# B&R Automation Studio project TD52 (part 13)

### fintrf.h
```c
#if defined(WITH_COMMENTS)
/*
 * fintrf.h	- MATLAB/FORTRAN interface header file. This file
 *		  contains the declaration of the pointer type needed
 *		  by the MATLAB/FORTRAN interface.
 *
 * Copyright 1984-2008 The MathWorks, Inc.
 * All Rights Reserved.
 */
#endif
#if defined(__x86_64__) || defined(_M_AMD64) || defined(__amd64) || \
    defined(__sparcv9)  || defined(__ppc64__)
# define mwpointer integer*8
# define mwPointer integer*8
# define MWPOINTER INTEGER*8
#else
# define mwpointer integer*4
# define mwPointer integer*4
# define MWPOINTER INTEGER*4
#endif

#if defined(MX_COMPAT_32)
# define mwsize  integer*4
# define mwSize  integer*4
# define MWSIZE  INTEGER*4
# define mwindex integer*4
# define mwIndex integer*4
# define MWINDEX INTEGER*4
# define mwsignedindex integer*4
# define mwSignedIndex integer*4
# define MWSIGNEDINDEX INTEGER*4
#else
# define mwsize  mwpointer
# define mwSize  mwpointer
# define MWSIZE  MWPOINTER
# define mwindex mwpointer
# define mwIndex mwpointer
# define MWINDEX MWPOINTER
# define mwsignedindex mwpointer
# define mwSignedIndex mwpointer
# define MWSIGNEDINDEX MWPOINTER
#endif

#if defined(WITH_COMMENTS)
/*
 * Compatibility layer for MEX files using the 32-bit mxArray APIs
 */
#endif

#if defined(MX_COMPAT_32)

#define mxCalcSingleSubscript mxCalcSingleSubscript700
#define mxCreateCellArray mxCreateCellArray700
#define mxCreateCellMatrix mxCreateCellMatrix700
#define mxCreateCharArray mxCreateCharArray700
#define mxCreateCharMatrixFromStrings mxCreateCharMatrixFromStrs700
#define mxCreateDoubleMatrix mxCreateDoubleMatrix700
#define mxCreateNumericArray mxCreateNumericArray700
#define mxCreateNumericMatrix mxCreateNumericMatrix700
#define mxCreateSparse mxCreateSparse700
#define mxCreateStructArray mxCreateStructArray700
#define mxCreateStructMatrix mxCreateStructMatrix700
#define mxGetCell mxGetCell700
#define mxGetDimensions mxGetDimensions700
#define mxGetField mxGetField700
#define mxGetFieldByNumber mxGetFieldByNumber700
#define mxGetProperty mxGetProperty700
#define mxGetIr mxGetIr700
#define mxGetJc mxGetJc700
#define mxGetNumberOfDimensions mxGetNumberOfDimensions700
#define mxGetNzmax mxGetNzmax700
#define mxGetString mxGetString700
#define mxSetCell mxSetCell700
#define mxSetDimensions mxSetDimensions700
#define mxSetField mxSetField700
#define mxSetFieldByNumber mxSetFieldByNumber700
#define mxSetProperty mxSetProperty700
#define mxSetIr mxSetIr700
#define mxSetJc mxSetJc700
#define mxSetM mxSetM700
#define mxSetN mxSetN700
#define mxSetNzmax mxSetNzmax700
#define mxGetM mxGetM700
#define mxGetN mxGetN700
#define mxGetNumberOfElements mxGetNumberOfElements700
#define mxGetElementSize mxGetElementSize700
#define mxMalloc mxMalloc700
#define mxCalloc mxCalloc700
#define mxRealloc mxRealloc700
#define mxCopyReal4ToPtr mxCopyReal4ToPtr700
#define mxCopyPtrToReal4 mxCopyPtrToReal4700
#define mxCopyReal8ToPtr mxCopyReal8ToPtr700
#define mxCopyPtrToReal8 mxCopyPtrToReal8700
#define mxCopyCharacterToPtr mxCopyCharacterToPtr700
#define mxCopyPtrToCharacter mxCopyPtrToCharacter700
#define mxCopyInteger1ToPtr mxCopyInteger1ToPtr700
#define mxCopyPtrToInteger1 mxCopyPtrToInteger1700
#define mxCopyInteger2ToPtr mxCopyInteger2ToPtr700
#define mxCopyPtrToInteger2 mxCopyPtrToInteger2700
#define mxCopyInteger4ToPtr mxCopyInteger4ToPtr700
#define mxCopyPtrToInteger4 mxCopyPtrToInteger4700
#define mxCopyInteger8ToPtr mxCopyInteger8ToPtr700
#define mxCopyPtrToInteger8 mxCopyPtrToInteger8700
#define mxCopyPtrToPtrArray mxCopyPtrToPtrArray700
#define mxCopyComplex16ToPtr mxCopyComplex16ToPtr700
#define mxCopyPtrToComplex16 mxCopyPtrToComplex16700
#define mxCopyComplex8ToPtr mxCopyComplex8ToPtr700
#define mxCopyPtrToComplex8 mxCopyPtrToComplex8700
#define mxCopyMWIndexToPtr mxCopyMWIndexToPtr700
#define mxCopyPtrToMWIndex mxCopyPtrToMWIndex700
#define mxCreateCharMatrixFromStrs mxCreateCharMatrixFromStrs700
#define MXCALCSINGLESUBSCRIPT MXCALCSINGLESUBSCRIPT700
#define MXCREATECELLARRAY MXCREATECELLARRAY700
#define MXCREATECELLMATRIX MXCREATECELLMATRIX700
#define MXCREATECHARARRAY MXCREATECHARARRAY700
#define MXCREATECHARMATRIXFROMSTRINGS MXCREATECHARMATRIXFROMSTRS700
#define MXCREATEDOUBLEMATRIX MXCREATEDOUBLEMATRIX700
#define MXCREATENUMERICARRAY MXCREATENUMERICARRAY700
#define MXCREATENUMERICMATRIX MXCREATENUMERICMATRIX700
#define MXCREATESPARSE MXCREATESPARSE700
#define MXCREATESTRUCTARRAY MXCREATESTRUCTARRAY700
#define MXCREATESTRUCTMATRIX MXCREATESTRUCTMATRIX700
#define MXGETCELL MXGETCELL700
#define MXGETDIMENSIONS MXGETDIMENSIONS700
#define MXGETFIELD MXGETFIELD700
#define MXGETFIELDBYNUMBER MXGETFIELDBYNUMBER700
#define MXGETPROPERTY MXGETPROPERTY700
#define MXGETIR MXGETIR700
#define MXGETJC MXGETJC700
#define MXGETNUMBEROFDIMENSIONS MXGETNUMBEROFDIMENSIONS700
#define MXGETNZMAX MXGETNZMAX700
#define MXGETSTRING MXGETSTRING700
#define MXSETCELL MXSETCELL700
#define MXSETDIMENSIONS MXSETDIMENSIONS700
#define MXSETFIELD MXSETFIELD700
#define MXSETFIELDBYNUMBER MXSETFIELDBYNUMBER700
#define MXSETPROPERTY MXSETPROPERTY700
#define MXSETIR MXSETIR700
#define MXSETJC MXSETJC700
#define MXSETM MXSETM700
#define MXSETN MXSETN700
#define MXSETNZMAX MXSETNZMAX700
#define MXGETM MXGETM700
#define MXGETN MXGETN700
#define MXGETNUMBEROFELEMENTS MXGETNUMBEROFELEMENTS700
#define MXGETELEMENTSIZE MXGETELEMENTSIZE700
#define MXMALLOC MXMALLOC700
#define MXCALLOC MXCALLOC700
#define MXREALLOC MXREALLOC700
#define MXCOPYREAL4TOPTR MXCOPYREAL4TOPTR700
#define MXCOPYPTRTOREAL4 MXCOPYPTRTOREAL4700
#define MXCOPYREAL8TOPTR MXCOPYREAL8TOPTR700
#define MXCOPYPTRTOREAL8 MXCOPYPTRTOREAL8700
#define MXCOPYCHARACTERTOPTR MXCOPYCHARACTERTOPTR700
#define MXCOPYPTRTOCHARACTER MXCOPYPTRTOCHARACTER700
#define MXCOPYINTEGER1TOPTR MXCOPYINTEGER1TOPTR700
#define MXCOPYPTRTOINTEGER1 MXCOPYPTRTOINTEGER1700
#define MXCOPYINTEGER2TOPTR MXCOPYINTEGER2TOPTR700
#define MXCOPYPTRTOINTEGER2 MXCOPYPTRTOINTEGER2700
#define MXCOPYINTEGER4TOPTR MXCOPYINTEGER4TOPTR700
#define MXCOPYPTRTOINTEGER4 MXCOPYPTRTOINTEGER4700
#define MXCOPYINTEGER8TOPTR MXCOPYINTEGER8TOPTR700
#define MXCOPYPTRTOINTEGER8 MXCOPYPTRTOINTEGER8700
#define MXCOPYPTRTOPTRARRAY MXCOPYPTRTOPTRARRAY700
#define MXCOPYCOMPLEX16TOPTR MXCOPYCOMPLEX16TOPTR700
#define MXCOPYPTRTOCOMPLEX16 MXCOPYPTRTOCOMPLEX16700
#define MXCOPYCOMPLEX8TOPTR MXCOPYCOMPLEX8TOPTR700
#define MXCOPYPTRTOCOMPLEX8 MXCOPYPTRTOCOMPLEX8700
#define MXCOPYMWINDEXTOPTR MXCOPYMWINDEXTOPTR700
#define MXCOPYPTRTOMWINDEX MXCOPYPTRTOMWINDEX700
#define MXCREATECHARMATRIXFROMSTRS MXCREATECHARMATRIXFROMSTRS700
#define mxcalcsinglesubscript mxcalcsinglesubscript700
#define mxcreatecellarray mxcreatecellarray700
#define mxcreatecellmatrix mxcreatecellmatrix700
#define mxcreatechararray mxcreatechararray700
#define mxcreatecharmatrixfromstrings mxcreatecharmatrixfromstrs700
#define mxcreatedoublematrix mxcreatedoublematrix700
#define mxcreatenumericarray mxcreatenumericarray700
#define mxcreatenumericmatrix mxcreatenumericmatrix700
#define mxcreatesparse mxcreatesparse700
#define mxcreatestructarray mxcreatestructarray700
#define mxcreatestructmatrix mxcreatestructmatrix700
#define mxgetcell mxgetcell700
#define mxgetdimensions mxgetdimensions700
#define mxgetfield mxgetfield700
#define mxgetfieldbynumber mxgetfieldbynumber700
#define mxgetproperty mxgetproperty700
#define mxgetir mxgetir700
#define mxgetjc mxgetjc700
#define mxgetnumberofdimensions mxgetnumberofdimensions700
#define mxgetnzmax mxgetnzmax700
#define mxgetstring mxgetstring700
#define mxsetcell mxsetcell700
#define mxsetdimensions mxsetdimensions700
#define mxsetfield mxsetfield700
#define mxsetfieldbynumber mxsetfieldbynumber700
#define mxsetproperty mxsetproperty700
#define mxsetir mxsetir700
#define mxsetjc mxsetjc700
#define mxsetm mxsetm700
#define mxsetn mxsetn700
#define mxsetnzmax mxsetnzmax700
#define mxgetm mxgetm700
#define mxgetn mxgetn700
#define mxgetnumberofelements mxgetnumberofelements700
#define mxgetelementsize mxgetelementsize700
#define mxmalloc mxmalloc700
#define mxcalloc mxcalloc700
#define mxrealloc mxrealloc700
#define mxcopyreal4toptr mxcopyreal4toptr700
#define mxcopyptrtoreal4 mxcopyptrtoreal4700
#define mxcopyreal8toptr mxcopyreal8toptr700
#define mxcopyptrtoreal8 mxcopyptrtoreal8700
#define mxcopycharactertoptr mxcopycharactertoptr700
#define mxcopyptrtocharacter mxcopyptrtocharacter700
#define mxcopyinteger1toptr mxcopyinteger1toptr700
#define mxcopyptrtointeger1 mxcopyptrtointeger1700
#define mxcopyinteger2toptr mxcopyinteger2toptr700
#define mxcopyptrtointeger2 mxcopyptrtointeger2700
#define mxcopyinteger4toptr mxcopyinteger4toptr700
#define mxcopyptrtointeger4 mxcopyptrtointeger4700
#define mxcopyinteger8toptr mxcopyinteger8toptr700
#define mxcopyptrtointeger8 mxcopyptrtointeger8700
#define mxcopyptrtoptrarray mxcopyptrtoptrarray700
#define mxcopycomplex16toptr mxcopycomplex16toptr700
#define mxcopyptrtocomplex16 mxcopyptrtocomplex16700
#define mxcopycomplex8toptr mxcopycomplex8toptr700
#define mxcopyptrtocomplex8 mxcopyptrtocomplex8700
#define mxcopymwindextoptr mxcopymwindextoptr700
#define mxcopyptrtomwindex mxcopyptrtomwindex700
#define mxcreatecharmatrixfromstrs mxcreatecharmatrixfromstrs700

#else

#ifndef __linux
#define mxCalcSingleSubscript mxCalcSingleSubscript730
#define mxCreateCellArray mxCreateCellArray730
#define mxCreateCellMatrix mxCreateCellMatrix730
#define mxCreateCharArray mxCreateCharArray730
#define mxCreateCharMatrixFromStrings mxCreateCharMatrixFromStrs730
#define mxCreateDoubleMatrix mxCreateDoubleMatrix730
#define mxCreateNumericArray mxCreateNumericArray730
#define mxCreateNumericMatrix mxCreateNumericMatrix730
#define mxCreateSparse mxCreateSparse730
#define mxCreateStructArray mxCreateStructArray730
#define mxCreateStructMatrix mxCreateStructMatrix730
#define mxGetCell mxGetCell730
#define mxGetDimensions mxGetDimensions730
#define mxGetField mxGetField730
#define mxGetFieldByNumber mxGetFieldByNumber730
#define mxGetProperty mxGetProperty730
#define mxGetIr mxGetIr730
#define mxGetJc mxGetJc730
#define mxGetNumberOfDimensions mxGetNumberOfDimensions730
#define mxGetNzmax mxGetNzmax730
#define mxGetString mxGetString730
#define mxSetCell mxSetCell730
#define mxSetDimensions mxSetDimensions730
#define mxSetField mxSetField730
#define mxSetFieldByNumber mxSetFieldByNumber730
#define mxSetProperty mxSetProperty730
#define mxSetIr mxSetIr730
#define mxSetJc mxSetJc730
#define mxSetM mxSetM730
#define mxSetN mxSetN730
#define mxSetNzmax mxSetNzmax730
#define mxGetM mxGetM730
#define mxGetN mxGetN730
#define mxGetNumberOfElements mxGetNumberOfElements730
#define mxGetElementSize mxGetElementSize730
#define mxMalloc mxMalloc730
#define mxCalloc mxCalloc730
#define mxRealloc mxRealloc730
#define mxCopyReal4ToPtr mxCopyReal4ToPtr730
#define mxCopyPtrToReal4 mxCopyPtrToReal4730
#define mxCopyReal8ToPtr mxCopyReal8ToPtr730
#define mxCopyPtrToReal8 mxCopyPtrToReal8730
#define mxCopyCharacterToPtr mxCopyCharacterToPtr730
#define mxCopyPtrToCharacter mxCopyPtrToCharacter730
#define mxCopyInteger1ToPtr mxCopyInteger1ToPtr730
#define mxCopyPtrToInteger1 mxCopyPtrToInteger1730
#define mxCopyInteger2ToPtr mxCopyInteger2ToPtr730
#define mxCopyPtrToInteger2 mxCopyPtrToInteger2730
#define mxCopyInteger4ToPtr mxCopyInteger4ToPtr730
#define mxCopyPtrToInteger4 mxCopyPtrToInteger4730
#define mxCopyInteger8ToPtr mxCopyInteger8ToPtr730
#define mxCopyPtrToInteger8 mxCopyPtrToInteger8730
#define mxCopyPtrToPtrArray mxCopyPtrToPtrArray730
#define mxCopyComplex16ToPtr mxCopyComplex16ToPtr730
#define mxCopyPtrToComplex16 mxCopyPtrToComplex16730
#define mxCopyComplex8ToPtr mxCopyComplex8ToPtr730
#define mxCopyPtrToComplex8 mxCopyPtrToComplex8730
#define mxCopyMWIndexToPtr mxCopyMWIndexToPtr730
#define mxCopyPtrToMWIndex mxCopyPtrToMWIndex730
#define mxCreateCharMatrixFromStrs mxCreateCharMatrixFromStrs730
#define MXCALCSINGLESUBSCRIPT MXCALCSINGLESUBSCRIPT730
#define MXCREATECELLARRAY MXCREATECELLARRAY730
#define MXCREATECELLMATRIX MXCREATECELLMATRIX730
#define MXCREATECHARARRAY MXCREATECHARARRAY730
#define MXCREATECHARMATRIXFROMSTRINGS MXCREATECHARMATRIXFROMSTRS730
#define MXCREATEDOUBLEMATRIX MXCREATEDOUBLEMATRIX730
#define MXCREATENUMERICARRAY MXCREATENUMERICARRAY730
#define MXCREATENUMERICMATRIX MXCREATENUMERICMATRIX730
#define MXCREATESPARSE MXCREATESPARSE730
#define MXCREATESTRUCTARRAY MXCREATESTRUCTARRAY730
#define MXCREATESTRUCTMATRIX MXCREATESTRUCTMATRIX730
#define MXGETCELL MXGETCELL730
#define MXGETDIMENSIONS MXGETDIMENSIONS730
#define MXGETFIELD MXGETFIELD730
#define MXGETFIELDBYNUMBER MXGETFIELDBYNUMBER730
#define MXGETPROPERTY MXGETPROPERTY730
#define MXGETIR MXGETIR730
#define MXGETJC MXGETJC730
#define MXGETNUMBEROFDIMENSIONS MXGETNUMBEROFDIMENSIONS730
#define MXGETNZMAX MXGETNZMAX730
#define MXGETSTRING MXGETSTRING730
#define MXSETCELL MXSETCELL730
#define MXSETDIMENSIONS MXSETDIMENSIONS730
#define MXSETFIELD MXSETFIELD730
#define MXSETFIELDBYNUMBER MXSETFIELDBYNUMBER730
#define MXSETPROPERTY MXSETPROPERTY730
#define MXSETIR MXSETIR730
#define MXSETJC MXSETJC730
#define MXSETM MXSETM730
#define MXSETN MXSETN730
#define MXSETNZMAX MXSETNZMAX730
#define MXGETM MXGETM730
#define MXGETN MXGETN730
#define MXGETNUMBEROFELEMENTS MXGETNUMBEROFELEMENTS730
#define MXGETELEMENTSIZE MXGETELEMENTSIZE730
#define MXMALLOC MXMALLOC730
#define MXCALLOC MXCALLOC730
#define MXREALLOC MXREALLOC730
#define MXCOPYREAL4TOPTR MXCOPYREAL4TOPTR730
#define MXCOPYPTRTOREAL4 MXCOPYPTRTOREAL4730
#define MXCOPYREAL8TOPTR MXCOPYREAL8TOPTR730
#define MXCOPYPTRTOREAL8 MXCOPYPTRTOREAL8730
#define MXCOPYCHARACTERTOPTR MXCOPYCHARACTERTOPTR730
#define MXCOPYPTRTOCHARACTER MXCOPYPTRTOCHARACTER730
#define MXCOPYINTEGER1TOPTR MXCOPYINTEGER1TOPTR730
#define MXCOPYPTRTOINTEGER1 MXCOPYPTRTOINTEGER1730
#define MXCOPYINTEGER2TOPTR MXCOPYINTEGER2TOPTR730
#define MXCOPYPTRTOINTEGER2 MXCOPYPTRTOINTEGER2730
#define MXCOPYINTEGER4TOPTR MXCOPYINTEGER4TOPTR730
#define MXCOPYPTRTOINTEGER4 MXCOPYPTRTOINTEGER4730
#define MXCOPYINTEGER8TOPTR MXCOPYINTEGER8TOPTR730
#define MXCOPYPTRTOINTEGER8 MXCOPYPTRTOINTEGER8730
#define MXCOPYPTRTOPTRARRAY MXCOPYPTRTOPTRARRAY730
#define MXCOPYCOMPLEX16TOPTR MXCOPYCOMPLEX16TOPTR730
#define MXCOPYPTRTOCOMPLEX16 MXCOPYPTRTOCOMPLEX16730
#define MXCOPYCOMPLEX8TOPTR MXCOPYCOMPLEX8TOPTR730
#define MXCOPYPTRTOCOMPLEX8 MXCOPYPTRTOCOMPLEX8730
#define MXCOPYMWINDEXTOPTR MXCOPYMWINDEXTOPTR730
#define MXCOPYPTRTOMWINDEX MXCOPYPTRTOMWINDEX730
#define MXCREATECHARMATRIXFROMSTRS MXCREATECHARMATRIXFROMSTRS730
#define mxcalcsinglesubscript mxcalcsinglesubscript730
#define mxcreatecellarray mxcreatecellarray730
#define mxcreatecellmatrix mxcreatecellmatrix730
#define mxcreatechararray mxcreatechararray730
#define mxcreatecharmatrixfromstrings mxcreatecharmatrixfromstrs730
#define mxcreatedoublematrix mxcreatedoublematrix730
#define mxcreatenumericarray mxcreatenumericarray730
#define mxcreatenumericmatrix mxcreatenumericmatrix730
#define mxcreatesparse mxcreatesparse730
#define mxcreatestructarray mxcreatestructarray730
#define mxcreatestructmatrix mxcreatestructmatrix730
#define mxgetcell mxgetcell730
#define mxgetdimensions mxgetdimensions730
#define mxgetfield mxgetfield730
#define mxgetfieldbynumber mxgetfieldbynumber730
#define mxgetproperty mxgetproperty730
#define mxgetir mxgetir730
#define mxgetjc mxgetjc730
#define mxgetnumberofdimensions mxgetnumberofdimensions730
#define mxgetnzmax mxgetnzmax730
#define mxgetstring mxgetstring730
#define mxsetcell mxsetcell730
#define mxsetdimensions mxsetdimensions730
#define mxsetfield mxsetfield730
#define mxsetfieldbynumber mxsetfieldbynumber730
#define mxsetproperty mxsetproperty730
#define mxsetir mxsetir730
#define mxsetjc mxsetjc730
#define mxsetm mxsetm730
#define mxsetn mxsetn730
#define mxsetnzmax mxsetnzmax730
#define mxgetm mxgetm730
#define mxgetn mxgetn730
#define mxgetnumberofelements mxgetnumberofelements730
#define mxgetelementsize mxgetelementsize730
#define mxmalloc mxmalloc730
#define mxcalloc mxcalloc730
#define mxrealloc mxrealloc730
#define mxcopyreal4toptr mxcopyreal4toptr730
#define mxcopyptrtoreal4 mxcopyptrtoreal4730
#define mxcopyreal8toptr mxcopyreal8toptr730
#define mxcopyptrtoreal8 mxcopyptrtoreal8730
#define mxcopycharactertoptr mxcopycharactertoptr730
#define mxcopyptrtocharacter mxcopyptrtocharacter730
#define mxcopyinteger1toptr mxcopyinteger1toptr730
#define mxcopyptrtointeger1 mxcopyptrtointeger1730
#define mxcopyinteger2toptr mxcopyinteger2toptr730
#define mxcopyptrtointeger2 mxcopyptrtointeger2730
#define mxcopyinteger4toptr mxcopyinteger4toptr730
#define mxcopyptrtointeger4 mxcopyptrtointeger4730
#define mxcopyinteger8toptr mxcopyinteger8toptr730
#define mxcopyptrtointeger8 mxcopyptrtointeger8730
#define mxcopyptrtoptrarray mxcopyptrtoptrarray730
#define mxcopycomplex16toptr mxcopycomplex16toptr730
#define mxcopyptrtocomplex16 mxcopyptrtocomplex16730
#define mxcopycomplex8toptr mxcopycomplex8toptr730
#define mxcopyptrtocomplex8 mxcopyptrtocomplex8730
#define mxcopymwindextoptr mxcopymwindextoptr730
#define mxcopyptrtomwindex mxcopyptrtomwindex730
#define mxcreatecharmatrixfromstrs mxcreatecharmatrixfromstrs730
#endif

#endif
```

### fixedpoint.h
```c
#include "fixpoint_spec.hpp"
/* Copyright 1994-2010 The MathWorks, Inc.
 * $Revision: 1.1.8.1 $
 * $Date: 2010/12/15 17:39:58 $
 */

#ifdef SUPPORTS_PRAGMA_ONCE
#pragma once
#endif

#ifndef fix_published_intro_h
#define fix_published_intro_h

/* Abstract:
 *
 * The primary motivation of this header file is to allow customers to
 * write C language S-functions that support fixed-point data types.  However,
 * the API in this header extends beyond fixed-point and includes support for
 * standard floating point and integer data types.
 *
 * This header contains definitions and prototypes for use in creating
 * Simulink S-functions that can process a wide variety of data types.
 * These data types include the Simulink builtin data types,
 *     double        single
 *     uint8         int8
 *     uint16        int16
 *     uint32        int32
 * all the MathWorks defined fixed-point data types such as
 *     sfix16_En15
 *     ufix32_En16
 *     ufix128
 *     sfix37_S3_B5
 * and the versions of data types obtained when Data Type Override is set
 * to Scaled Doubles such as
 *     flts16
 *     flts16_En15
 *     fltu32_S3_B5
 *
 * This header file contains functions and definitions that allow S-functions
 * to determine which of these data types an input port or output port is
 * using.  The S-function can also specify which of these data types should
 * be used for an input, output, DWork state, or Runtime Parameter.  The
 * information required to properly read to and write from different variables
 * of each data type is given.
 */

/* Note on License Design:
 *
 * The following comments are simply an attempt to clarify the License Design
 * so that authors can write better S-functions.
 * As of
 *      Release 13
 *      Simulink 5.0
 *      Fixed-Point Blockset 4.0
 * all the blocks from Fixed-Point Blockset were merged into Simulink.  All
 * the blocks are installed even if a user does not have a Fixed-Point License.
 * Simulink customers can use all the blocks with any builtin data types that a
 * block supports.  If all the blocks in a model are only using builtin data
 * types and the Min-Max-Overflow Logging Mode is set to Force Off, then a
 * Fixed-Point License is NOT required.  If any block in a model is "actively"
 * using a non-builtin fixed-point data type or is actively logging Min-Max and/or
 * Overflow information, then a Fixed-Point License will be required for the
 * remainder of that Matlab session.
 *   Even if blocks in a model are configured to have fixed-point signals and/or
 * configured to log Min-Max-Overflow information, then simply loading, viewing,
 * editing, or saving a model should not trigger active use.  Actions such as
 * Update Diagram, Simulation, and Code Generation from such a model are active
 * use and would cause a Fixed-Point License to be checked out.
 *   S-functions written using the API in this header file should be able to
 * follow this license design.  For example, suppose an S-function is written
 * so that it can handle any builtin or fixed-point data type.  Suppose in a
 * particular model, this S-function is processing just builtin data types such
 * as double, single, uint8, or int32.  That use case would not trigger a
 * Fixed-Point License to be checked out.  Suppose in a different model,
 * the S-function was processing non-builtin fixed-point data types.  That use,
 * like any other use of fixed-point data types, would cause a Fixed-Point
 * License to be checked out.
 *   The key pitfall S-function authors must guard against is registering
 * a fixed-point data type when a model is simply being loaded or viewed.  In
 * Simulink jargon, loading or opening a model or sub-system is a
 * "Sizes Call Only."  The Simulink S-function API provides a way to detect a
 * "Sizes Call Only", so by careful programming, an S-function author can avoid
 * Fixed-Point License problems when a user is simply loading or viewing a model.
 */

/* Simulink supports fixed-point data types with any number of bits from
 *    1 to FXP_MAX_BITS for unsigned numbers and
 *    2 to FXP_MAX_BITS for signed numbers.
 * The API in this header file treats pure integers just like
 * any other fixed-point numbers.  Pure integers just happen
 * to have trivial scaling.  The 6 standard Simulink integer
 * types uint8, int8, uint16, int16, uint32, and int32 are not
 * exceptions.  They are treated like fixed-point numbers
 * that happened to have trivial scaling and happened to have
 * 8, 16, or 32 bits.  The same API applies.
 *   Simulink builtin integers are special only in that they do
 * not trigger the need for a Fixed-Point License.
 *
 * The number of bits used to represent a signal in simulation
 * may be more than the number specified.  In this case, the
 * signals will be emulated inside various sized containers
 * according to the following rules.  For 32 or fewer bits, the
 * rules are simple.  For 32 or fewer bits, the container is a
 * scalar integer type directly understood by the compiler.  The
 * case of using a scalar integer type is classified as single-word.
 * The three cases with 32 or fewer bits are shown by a table.
 *
 *   Specified Bits       Container Bits   Container typedef
 *    1 to  8              8               int8_T  or uint8_T
 *    9 to 16             16               int16_T or uint16_T
 *   17 to 32             32               int32_T or uint32_T
 *
 * For 33 or more bits, the rules are more complicated and can
 * depend on the model, the Matlab Host, the current target
 * for code generation, and the version of Simulink Fixed Point
 * being used.  Signals with 33 or more bits will either be stored
 * using a single-word
 * container with more than 32 bits or will be stored using a
 * multi-word representation.
 *
 * All multi-word representations will follow a general form.
 *
 * typedef struct {
 *     SOME_UNSIGNED_CHUNK_TYPE chunks[ NUM_CHUNKS_FOR_M_BITS ];
 * } (u)intM_T
 *
 * The chunk at index zero will hold the least significant bits, and
 * the highest index will hold the most significant bits.
 *
 * Whether single-word or multi-word is used can depend on
 * the model, the Matlab Host, the current
 * target for code generation, and the version of Simulink Fixed Point.
 * The specific type used for SOME_UNSIGNED_CHUNK_TYPE can also vary depending
 * on the model, the Matlab Host, the current target for code generation,
 * and the version of Simulink Fixed Point.
 *
 * To be portable, sfunctions that are intended to support fixed-point
 * signals with more than 32 bits must react to container variations
 * at runtime.  The most general way to do this is to use the interfaces
 * for getting and setting "bit-regions" provided by this header.
 * To support use of code optimized to a specific additional APIs
 * are provided that can query the current properties of a data type.
 * However, sfunction authors need to be aware the properties of a data
 * type can vary depending on
 * the model, the Matlab Host, the current
 * target for code generation, and the version of Simulink Fixed Point.
 * A robustly written sfunction will need to check the properties at runtime
 * at least once after update diagram has started.  The most portable sfunctions
 * will be written so that they can use an optimized case if possible or
 * switch to general bit-region case if necessary.  At the very least,
 * a robust sfunction will need to gracefully set an error if does not
 * have a case that supports the current memory layout.  Keep in mind that
 * supporting every specific case for the current release of Simulink Fixed Point
 * does not guarantee that every specific case in a future release will be
 * covered.  For this reason, it is best to have bit-region case or at
 * the very least gracefully error if needed.
 *
 * For signed numbers, the bit encoding format is always
 * two's complement.
 *
 * When the specified number of bits is less than the size of
 * the container, the desired bits are always stored in the
 * least significant part of the container.  Any "unused" bits
 * are in the most significant part of the container.
 *
 * For both single word case and multiword cases, any unused bits
 * must be set to a sign extension.  If the data type is
 * an unsigned number, then obviously, the number is always
 * nonnegative so the (implicit) sign bit is zero.  For unsigned
 * data types, all unused bits must always be cleared to zero.
 *    If the data type is a signed number, then the sign bit is
 * one for strictly negative numbers and zero otherwise.  If
 * the stored integer is negative, then all unused bits must be
 * set to one.  If the stored integer is positive, then all
 * unused bits must be cleared to zero.
 *
 * Simulink also supports two builtin floating point data types.
 * These are the standard floating point singles and doubles.
 *
 * Simulink also supports a data type category that is a hybrid
 * between floating-point and fixed-point.  This category is
 * called ScaledDouble.  ScaledDouble cases occur when
 * an individual block is configured to have a fixed-point
 * output, but the system it lives in has its Data Type Override
 * setting for a system is set to Scaled Doubles.  The
 * resulting data type has the scaling the fixed-point
 * specification, but stores its output using floating
 * point doubles.  Storing in a double means that overflow
 * and precision issues are almost always eliminated. Removing the
 * range and precision issues is very useful for benchmarking, testing,
 * and debugging.
 *   ScaledDouble data types contain information
 * signedness and number of bits of what their non-overrided data
 * types would have been.  This is useful for information for other
 * portions of the model that are not being debugged with Data Type
 * Override.
 */

#endif /* fix_published_intro_h */
/* Copyright 1994-2010 The MathWorks, Inc.
 * $Revision: 1.1.6.1 $
 * $Date: 2010/06/15 00:02:53 $
 */

#ifdef SUPPORTS_PRAGMA_ONCE
#pragma once
#endif

#ifndef fxplimits_h
#define fxplimits_h

#define FXP_MAX_BITS 128

#endif /* fxplimits_h */
/* Copyright 1994-2010 The MathWorks, Inc.
 * $Revision: 1.1.6.1 $
 * $Date: 2010/06/15 00:02:51 $
 */

#ifdef SUPPORTS_PRAGMA_ONCE
#pragma once
#endif

#ifndef fxpchunkarrary_h
#define fxpchunkarrary_h

typedef uint32_T FXP_CHUNK_T;

#define FXP_BITS_PER_CHUNK 32

#define FXP_NUM_CHUNKS ( FXP_MAX_BITS / FXP_BITS_PER_CHUNK )

#define FXP_INDEX_LEAST_SIGNIFICANT_CHUNK 0

#define FXP_INDEX_MOST_SIGNIFICANT_CHUNK  ( FXP_NUM_CHUNKS - 1 )

#define FXP_ALL_ONES_CHUNK 0xFFFFFFFFul

typedef struct fxpChunkArray_tag
{
    FXP_CHUNK_T chunk[ FXP_NUM_CHUNKS ];

} fxpChunkArray;

#endif /* fxpchunkarrary_h */
/* Copyright 1994-2010 The MathWorks, Inc.
 * $Revision: 1.1.8.1 $
 * $Date: 2010/12/15 17:40:00 $
 */

#ifdef SUPPORTS_PRAGMA_ONCE
#pragma once
#endif

#ifndef fxpsimulinkscalingintro_h
#define fxpsimulinkscalingintro_h

/* Simulink Scaling
 *
 * Simulink data types support scaling.  The Fixed-Point User's Guide
 * presents the following general formula.
 *
 *    V = S * Q + B
 *
 * where
 *
 *    V is the Real World Value in the engineering units of choice
 *    Q is the called the Stored Integer Value.  It is the raw value
 *      stored in the digital hardware.  Despite the name Q can use
 *      an integer or a floating point format.
 *    S is the Slope.  For clarity, this is also called the Total-Slope
 *    B is the Bias
 *
 * The Total-Slope is often decomposed into two parts.
 *
 *    S = F * 2^E
 *
 * where
 *
 *   1. <= F < 2.0
 *
 *    F is the Fractional Slope
 *    E is the Fixed Exponent, E is always an integer.
 *
 * If
 *    B == 0.0
 * and
 *    F == 1.0
 * then
 * there is a clean binary point interpretation.
 *
 *    Fraction Length = -1 * Fixed Exponent
 *
 * For example, if
 *    S == 0.125
 *    B == 0.0
 * then
 *    F == 1.0
 *    E == -3
 * so
 *    Fraction Length = 3
 * therefore, this data type has 3 bits to the right of the
 * binary point.
 *
 * The concept of scaling is most useful for fixed-point cases, but
 * it does generalize to all the scalar numeric data types.  For
 * floating point doubles and singles and for pure integers,
 * the scaling is trivial
 *    B == 0
 *    S == 1
 *    F == 1
 *    E == 0
 *    Fraction Length == 0
 * The access methods to get scaling information can be used
 * for all the data types, they just return trivial values
 * when the scaling is trivial.
 */

#endif /* fxpsimulinkscalingintro_h */
/* Copyright 1994-2010 The MathWorks, Inc.
 * $Revision: 1.1.6.1 $
 * $Date: 2010/06/15 00:02:55 $
 */

#ifdef SUPPORTS_PRAGMA_ONCE
#pragma once
#endif

#ifndef fxpmodeoverflow_h
#define fxpmodeoverflow_h

/* The enums specify the overflow handling modes supported by most fixed-point
 * math functions.
 */
typedef enum fxpModeOverflow_tag {
  FXP_OVERFLOW_WRAP = 0, /* must be zero */
  FXP_OVERFLOW_SATURATE

} fxpModeOverflow;

#endif /* fxpmodeoverflow_h */
/* Copyright 1994-2010 The MathWorks, Inc.
 * $Revision: 1.1.6.1 $
 * $Date: 2010/06/15 00:02:57 $
 */

#ifdef SUPPORTS_PRAGMA_ONCE
#pragma once
#endif

#ifndef fxpmoderounding_h
#define fxpmoderounding_h

/* The enums specify the rounding modes supported by most fixed-point
 * math functions.
 */
typedef enum fxpModeRounding_tag {
  FXP_ROUND_ZERO = 0, /* must be zero */
  FXP_ROUND_NEAR,
  FXP_ROUND_CEIL,
  FXP_ROUND_FLOOR,
  FXP_ROUND_SIMPLEST,
  FXP_ROUND_NEAR_ML, /* Round -x.5 to -(x+1) not -x so as to match MATLAB. */
  FXP_ROUND_CONVERGENT
} fxpModeRounding;

#define FXP_ROUND_METHOD_COUNT ((FXP_ROUND_CONVERGENT)+1)

#endif /* fxpmoderounding_h */
/* Copyright 1994-2010 The MathWorks, Inc.
 * $Revision: 1.1.6.1 $
 * $Date: 2010/06/15 00:02:59 $
 */

#ifdef SUPPORTS_PRAGMA_ONCE
#pragma once
#endif

#ifndef fix_published_fxpOverflowLogs_h
#define fix_published_fxpOverflowLogs_h

/* Overflow logging structure
 *
 * Some fixed-point math functions accept a pointer to this structure.
 * These functions will initialize each of the event counts to zero.  Then
 * the functions will carryout the requested math operations.  Each
 * time an event is detect during the math operation the appropriate
 * count will be incremented.  The increment operations makes sure
 * the count does not overflow to zero; it will saturate to the upper limit.
 *
 * For example, suppose a fixed-point conversion function is called. Suppose,
 * one overflow occurred during the conversion.  After the function return,
 * the memory pointed to be overflow logging structure pointer would indicate
 * one overflow, zero saturations, and zero divide-by-zeros.
 */
typedef struct fxpOverflowLogs_tag
{
      int OverflowOccurred;
      int SaturationOccurred;
      int DivisionByZeroOccurred;

} fxpOverflowLogs;

#endif /* fix_published_fxpOverflowLogs_h */
/* Copyright 1994-2011 The MathWorks, Inc.
 *
 *
 */

#ifdef SUPPORTS_PRAGMA_ONCE
#pragma once
#endif

#ifndef fix_published_sfun_api_h
#define fix_published_sfun_api_h

/* Function: ssRegisterDataTypeFxpBinaryPoint ===============================
 *
 * This function fully registers a fixed-point data type with Simulink and
 * returns a Data Type Id.  Unlike the standard Simulink function,
 * ssRegisterDataType, additional registration steps do not need to be taken
 * and should not be taken.  The returned Data Type Id can be used to specify
 * the data types of input ports, output ports, RunTimeParameters, and DWork
 * states.  The Data Type Id can also be used with all the standard
 * data type access methods in simstruc.h such as ssGetDataTypeSize.
 *
 * The input arguments are
 *    isSigned              TRUE if signed, FALSE if unsigned
 *    wordLength            total number of bits including any sign bit
 *    fractionLength        number of bit to right of binary point
 *    obeyDataTypeOverride  if FALSE ignore system's setting for Data Type Override
 *                          if TRUE obey Data Type Override setting, depending
 *                          on Data Type Override, resulting data type could be
 *                          True Double, True Single, Scaled Double, or the
 *                          requested fixed point type.
 *
 * Cautions:
 *
 * 1) If the registered data type is not one of the builtin data types, then
 * a Fixed-Point License will be checked out.  To prevent, a Fixed-Point
 * License from being checked out when a user simply opens or views a model,
 * calls to registration should be protected with
 *    if ( ssGetSimMode(S) != SS_SIMMODE_SIZES_CALL_ONLY )
 *       ssRegisterDataType ...
 *
 * 2) There is no fixed relationship between the Data Type Id value and
 * the input arguments.  Simulink hands out data type Ids on a first come, first
 * served basis, so small changes to a model can cause the a different data
 * type id value to be returned.  Always uses functions to get data type
 * attributes from the data type id; never directly rely on the data type
 * id value.
 */
FIXPOINT_EXPORT_EXTERN_C DTypeId ssRegisterDataTypeFxpBinaryPoint(
    SimStruct *S,
    int isSigned,
    int wordLength,
    int fractionLength,
    int obeyDataTypeOverride
    );

/* Function: ssRegisterDataTypeFxpSlopeBias ===============================
 *
 * This function fully registers a fixed-point data type with Simulink and
 * returns a Data Type Id.  Unlike the standard Simulink function,
 * ssRegisterDataType, additional registration steps do not need to be taken
 * and should not be taken.  The returned Data Type Id can be used to specify
 * the data types of input ports, output ports, RunTimeParameters, and DWork
 * states.  The Data Type Id can also be used with all the standard
 * data type access methods in simstruc.h such as ssGetDataTypeSize.
 *
 * The input arguments are
 *    isSigned              TRUE if signed, FALSE if unsigned
 *    wordLength            total number of bits including any sign bit
 *    totalSlope            total slope
 *    bias                  bias
 *    obeyDataTypeOverride  if FALSE ignore system's setting for Data Type Override
 *                          if TRUE obey Data Type Override setting, depending
 *                          on Data Type Override, resulting data type could be
 *                          True Double, True Single, Scaled Double, or the
 *                          requested fixed point type.
 *
 * Cautions:
 *
 * 1) If the registered data type is not one of the builtin data types, then
 * a Fixed-Point License will be checked out.  To prevent, a Fixed-Point
 * License from being checked out when a user simply opens or views a model,
 * calls to registration should be protected with
 *    if ( ssGetSimMode(S) != SS_SIMMODE_SIZES_CALL_ONLY )
 *       ssRegisterDataType ...
 *
 * 2) There is no fixed relationship between the Data Type Id value and
 * the input arguments.  Simulink hands out data type Ids on a first come, first
 * served basis, so small changes to a model can cause the a different data
 * type id value to be returned.  Always uses functions to get data type
 * attributes from the data type id; never directly rely on the data type
 * id value.
 */
FIXPOINT_EXPORT_EXTERN_C DTypeId ssRegisterDataTypeFxpSlopeBias(
    SimStruct *S,
    int isSigned,
    int wordLength,
    double totalSlope,
    double bias,
    int obeyDataTypeOverride
    );

/* Function: ssRegisterDataTypeFxpFSlopeFixExpBias =============================
 *
 * This function fully registers a fixed-point data type with Simulink and
 * returns a Data Type Id.  Unlike the standard Simulink function,
 * ssRegisterDataType, additional registration steps do not need to be taken
 * and should not be taken.  The returned Data Type Id can be used to specify
 * the data types of input ports, output ports, RunTimeParameters, and DWork
 * states.  The Data Type Id can also be used with all the standard
 * data type access methods in simstruc.h such as ssGetDataTypeSize.
 *
 * The input arguments are
 *    isSigned              TRUE if signed, FALSE if unsigned
 *    wordLength            total number of bits including any sign bit
 *    fractionalSlope       fractional slope
 *    fixedExponent         fixed exponent
 *    bias                  bias
 *    obeyDataTypeOverride  if FALSE ignore system's setting for Data Type Override
 *                          if TRUE obey Data Type Override setting, depending
 *                          on Data Type Override, resulting data type could be
 *                          True Double, True Single, Scaled Double, or the
 *                          requested fixed point type.
 *
 * Cautions:
 *
 * 1) If the registered data type is not one of the builtin data types, then
 * a Fixed-Point License will be checked out.  To prevent, a Fixed-Point
 * License from being checked out when a user simply opens or views a model,
 * calls to registration should be protected with
 *    if ( ssGetSimMode(S) != SS_SIMMODE_SIZES_CALL_ONLY )
 *       ssRegisterDataType ...
 *
 * 2) There is no fixed relationship between the Data Type Id value and
 * the input arguments.  Simulink hands out data type Ids on a first come, first
 * served basis, so small changes to a model can cause the a different data
 * type id value to be returned.  Always uses functions to get data type
 * attributes from the data type id; never directly rely on the data type
 * id value.
 */
FIXPOINT_EXPORT_EXTERN_C DTypeId ssRegisterDataTypeFxpFSlopeFixExpBias(
    SimStruct *S,
    int isSigned,
    int wordLength,
    double fractionalSlope,
    int fixedExponent,
    double bias,
    int obeyDataTypeOverride
    );

/* Function: ssRegisterDataTypeFxpScaledDouble =============================
 *
 * This function fully registers a fixed-point data type with Simulink and
 * returns a Data Type Id.  Unlike the standard Simulink function,
 * ssRegisterDataType, additional registration steps do not need to be taken
 * and should not be taken.  The returned Data Type Id can be used to specify
 * the data types of input ports, output ports, RunTimeParameters, and DWork
 * states.  The Data Type Id can also be used with all the standard
 * data type access methods in simstruc.h such as ssGetDataTypeSize.
 *
 * The input arguments are
 *    isSigned              TRUE if signed, FALSE if unsigned
 *    wordLength            total number of bits including any sign bit
 *    fractionalSlope       fractional slope
 *    fixedExponent         fixed exponent
 *    bias                  bias
 *    obeyDataTypeOverride  if FALSE ignore system's setting for Data Type Override
 *                          if TRUE obey Data Type Override setting, depending
 *                          on Data Type Override, resulting data type could be
 *                          True Double, True Single, Scaled Double, or the
 *                          requested fixed point type.
 *
 * Cautions:
 *
 * 1) If the registered data type is not one of the builtin data types, then
 * a Fixed-Point License will be checked out.  To prevent, a Fixed-Point
 * License from being checked out when a user simply opens or views a model,
 * calls to registration should be protected with
 *    if ( ssGetSimMode(S) != SS_SIMMODE_SIZES_CALL_ONLY )
 *       ssRegisterDataType ...
 *
 * 2) There is no fixed relationship between the Data Type Id value and
 * the input arguments.  Simulink hands out data type Ids on a first come, first
 * served basis, so small changes to a model can cause the a different data
 * type id value to be returned.  Always uses functions to get data type
 * attributes from the data type id; never directly rely on the data type
 * id value.
 */
FIXPOINT_EXPORT_EXTERN_C DTypeId ssRegisterDataTypeFxpScaledDouble(
    SimStruct *S,
    int isSigned,
    int wordLength,
    double fractionalSlope,
    int fixedExponent,
    double bias,
    int obeyDataTypeOverride
    );

/* Function: ssGetDataTypeIsFxpFltApiCompat ==============================
 *
 * Giving a registered Data Type Id as input, determine if it is
 * supported by the API for user written fixed-point and floating-point
 * s-functions.  Support covers all the standard Simulink numeric types
 * double, single, uint8, ..., int32.  It also includes all the Fixed-Point
 * data types, including ScaledDouble versions.
 */
FIXPOINT_EXPORT_EXTERN_C int ssGetDataTypeIsFxpFltApiCompat(
    SimStruct *S,
    DTypeId dataTypeId
    );

typedef enum fxpStorageContainerCategory_tag {
    FXP_STORAGE_UNKNOWN = 0,
    FXP_STORAGE_DOUBLE,
    FXP_STORAGE_SINGLE,
    FXP_STORAGE_UINT8,
    FXP_STORAGE_INT8,
    FXP_STORAGE_UINT16,
    FXP_STORAGE_INT16,
    FXP_STORAGE_UINT32,
    FXP_STORAGE_INT32,
    FXP_STORAGE_CHUNKARRAY,
    FXP_STORAGE_SCALEDDOUBLE,
    FXP_STORAGE_OTHER_SINGLE_WORD,
    FXP_STORAGE_MULTIWORD
} fxpStorageContainerCategory;

/* Function: ssGetDataTypeStorageContainCat ===============================
 *
 * Giving a registered Data Type Id as input, determine the Storage Container
 * Category used to represent Input Signals, Output Signals, Run Time
 * Parameters, DWorks, etc. during Simulink Simulations.
 *   Descriptions of the Storage Containers and the definitions of
 * the output fxpStorageContainerCategory are given earlier in this header
 * file.
 *   This function will error out if ssGetDataTypeIsFxpFltApiCompat
 * returns false.
 */
FIXPOINT_EXPORT_EXTERN_C fxpStorageContainerCategory ssGetDataTypeStorageContainCat(
    SimStruct *S,
    DTypeId dataTypeId
    );

/* Function: ssGetDataTypeStorageContainSize ===============================
 *
 * Giving a registered Data Type Id as input, determine the Storage Container
 * Size used to represent Input Signals, Output Signals, Run Time
 * Parameters, DWorks, etc. during Simulink Simulations.  This is the size
 * that the sizeof() function would return.  This is the appropriate size
 * measurement to pass to functions like memcpy().
 *   This function will error out if ssGetDataTypeIsFxpFltApiCompat
 * returns false.
 *
 * This functions gives the same answer as the standard function
 * ssGetDataTypeSize.  This alternate version is only provide to reinforce
 * the distinction between specified word length and container size.  For
 * example, sfix24_En10 is specified to have 24 bits, but it actually is
 * stored in a larger container during Simulink Simulations.  The size of
 * the larger container is returned by this function.  This is the proper
 * value to use for memcpy, malloc, etc.
 */
FIXPOINT_EXPORT_EXTERN_C size_t ssGetDataTypeStorageContainerSize(
    SimStruct *S,
    DTypeId dataTypeId
    );

/* Function: ssGetDataTypeIsFixedPoint ===============================
 *
 * Giving a registered Data Type Id as input, determine the if the data
 * type is a fixed-point type.  Pure integers including the standard Simulink
 * integer types uint8, int8, uint16, uint32, and int32 are classified
 * as fixed-point types by this function.  Double, Single, and
 * ScaledDouble are NOT classified as fixed-point types.
 *   This function will error out if ssGetDataTypeIsFxpFltApiCompat
 * returns false.
 */
FIXPOINT_EXPORT_EXTERN_C int ssGetDataTypeIsFixedPoint(
    SimStruct *S,
    DTypeId dataTypeId
    );

/* Function: ssGetDataTypeIsFloatingPoint ===============================
 *
 * Giving a registered Data Type Id as input, determine the if the data
 * type is a true floating-point type.  Double and Single are true floating-
 * point types.  ScaledDouble is NOT classified as true float-point.
 *   This function will error out if ssGetDataTypeIsFxpFltApiCompat
 * returns false.
 */
FIXPOINT_EXPORT_EXTERN_C int ssGetDataTypeIsFloatingPoint(
    SimStruct *S,
    DTypeId dataTypeId
    );

/* Function: ssGetDataTypeFxpWordLength ===============================
 *
 * Giving a registered Data Type Id as input, determine the word length
 * of the data type.
 *     When the data type is fixed-point (including pure
 * integers), the word length is the total number of bits including
 * any sign bits, any bits in the integer part, and any bits in the
 * fractional bits.
 *     When the data type is ScaledDouble, the
 * word length is the total bits the original data type would have
 * used if override had not occurred.  For example, flts32_En4 would
 * have been sfix32_En4 if Data Type Override was off.  The word length is
 * therefore 32 bits.
 *     When the data type is true floating-point, this function errors
 * out.  Word length for a floating-point data type can mean different
 * things to different users.  For some, word length should only be the
 * physical mantissa bits excluding the hidden lead one.  For others,
 * the hidden leading one should be included.  For still others, the
 * word length should be all the physical bits including sign bit,
 * exponent bits, and mantissa bits, but not the hidden bit.  Rather
 * than mislead some users, this function errors out.
 *   This function will error out if ssGetDataTypeIsFxpFltApiCompat
 * returns false.
 */
FIXPOINT_EXPORT_EXTERN_C int ssGetDataTypeFxpWordLength(
    SimStruct *S,
    DTypeId dataTypeId
    );

/* Function: ssGetDataTypeFxpContainWordLen ===============================
 *
 * Giving a registered Data Type Id as input, determine the word length
 * of the storage container.
 *    When the data type is fixed-point (including pure
 * integers), the word length is the total number of bits including
 * any sign bits, any bits in the integer part, and any bits in the
 * fractional bits.
 *   The information provided by this function is not meaning full
 * when the data type is ScaledDouble or true floating point.  For
 * these data types, this function will error out.
 *   This function will error out if ssGetDataTypeIsFxpFltApiCompat
 * returns false.
 */
FIXPOINT_EXPORT_EXTERN_C int ssGetDataTypeFxpContainWordLen(
    SimStruct *S,
    DTypeId dataTypeId
    );

/* Function: ssGetDataTypeFxpIsSigned ===============================
 *
 * Giving a registered Data Type Id as input, return true if the data
 * type is signed, and return false if it is unsigned.
 *    When the data type is fixed-point (including pure
 * integers), the meaning of signed or unsigned is obvious.
 *     When the data type is ScaledDouble, the whether the data type
 * is signed or unsigned is determined by what the original data type would
 * have used if override had not occurred.  For example, flts32_En4 would
 * have been sfix32_En4 if Data Type Override was off.  This uses a signed
 * integer so the return value is true.  Conversely, fltu8_S3 would have
 * used ufix8_S3 which is unsigned, so false would be returned.
 *     When the data type is true floating-point, this function errors
 * out.  Asking whether a floating point number is signed or unsigned causes
 * some confusion, so this is prevented.
 *   This function will error out if ssGetDataTypeIsFxpFltApiCompat
 * returns false.
 */
FIXPOINT_EXPORT_EXTERN_C int ssGetDataTypeFxpIsSigned(
    SimStruct *S,
    DTypeId dataTypeId
    );

/* Function: ssGetDataTypeIsScalingTrivial =============================
 *
 * Giving a registered Data Type Id as input, determine if the scaling
 * is the trivial case of
 *    Slope   S == 1.0
 *    Bias    B == 0.0
 * This is always true for pure integers like int8 and for the true floating
 * point types double and single.  It will also be true for ScaledDouble
 * of pure integers such as flts8.  For binary point scaling, trivial means
 * the binary point is just to the right of the least significant bit.
 * Equivalently, the fraction length is zero.
 *   This function will error out if ssGetDataTypeIsFxpFltApiCompat
 * returns false.
 */
FIXPOINT_EXPORT_EXTERN_C int ssGetDataTypeIsScalingTrivial(
    SimStruct *S,
    DTypeId dataTypeId
    );

/* Function: ssGetDataTypeIsScalingPow2 ===========================
 *
 * Giving a registered Data Type Id as input, determine if the scaling
 * is an exact power of two
 *    Fractional Slope   F == 1.0
 *    Bias               B == 0.0
 * If the scaling is trivial, then the answer is true.  For fixed-point
 * cases, the answer is true if there is a clean binary point interpretation
 * of the scaling.
 *    Many fixed-point algorithms are only designed to handle power of
 * two scaling.  For this algorithms, this function can be called in
 * mdlSetInputPortDataType and mdlSetOutputPortDataType to prevent
 * unsupported data types from being accepted.
 *   This function will error out if ssGetDataTypeIsFxpFltApiCompat
 * returns false.
 */
FIXPOINT_EXPORT_EXTERN_C int ssGetDataTypeIsScalingPow2(
    SimStruct *S,
    DTypeId dataTypeId
    );

/* Function: ssGetDataTypeFractionLength ===============================
 *
 * Giving a registered Data Type Id as input, determine the fraction
 * length for data types that use power of two scaling.
 *    This function should be called only if ssGetDataTypeIsScalingPow2
 * returns true.  It errors out otherwise.
 *   This function will error out if ssGetDataTypeIsFxpFltApiCompat
 * returns false.
 */
FIXPOINT_EXPORT_EXTERN_C int ssGetDataTypeFractionLength(
    SimStruct *S,
    DTypeId dataTypeId
    );

/* Function: ssGetDataTypeTotalSlope ===============================
 *
 * Giving a registered Data Type Id as input, determine the scalings
 * total slope.
 *    S = F * 2^E
 * where
 *   1. <= F < 2.0
 *   S is the Total Slope
 *   F is the Fractional Slope
 *   E is the Fixed Exponent, E is always an integer
 *
 *     When the data type is ScaledDouble, the slope is determined by
 * what the original data type would  have used if override had not occurred.
 * For example, flts32_En4 would have been sfix32_En4 if Data Type Override was
 * off.  The total slope is 0.0625 = 2^-4.   For fltu16_S7p98, the total
 * slope is 7.98
 *     When the data type has trivial scaling, including floating point
 * double and single, the total slope is the trivial value 1.
 *   This function will error out if ssGetDataTypeIsFxpFltApiCompat
 * returns false.
 */
FIXPOINT_EXPORT_EXTERN_C double ssGetDataTypeTotalSlope(
    SimStruct *S,
    DTypeId dataTypeId
    );

/* Function: ssGetDataTypeBias ===============================
 *
 * Giving a registered Data Type Id as input, determine the scalings
 * bias.
 *     When the data type is ScaledDouble, the slope is determined by
 * what the original data type would  have used if override had not occurred.
 * For example, flts32_En4 would have been sfix32_En4 if Data Type Override was
 * off.  The bias is simply 0.   For fltu16_S3_Bn55p32, the total
 * slope is -55.32
 *     When the data type has trivial scaling, including floating point
 * double and single, the bias is the trivial value 0.  Likewise, when
 * the data type has power of two scaling, the bias is always the trivial
 * value 0.
 *   This function will error out if ssGetDataTypeIsFxpFltApiCompat
 * returns false.
 */
FIXPOINT_EXPORT_EXTERN_C double ssGetDataTypeBias(
    SimStruct *S,
    DTypeId dataTypeId
    );

/* Function: ssGetDataTypeFracSlope ===============================
 *
 * Giving a registered Data Type Id as input, determine the scalings
 * fractional slope.
 *    S = F * 2^E
 * where
 *   1. <= F < 2.0
 *   S is the Total Slope
 *   F is the Fractional Slope
 *   E is the Fixed Exponent, E is always an integer
 *
 *     When the data type is ScaledDouble, the slope is determined by
 * what the original data type would  have used if override had not occurred.
 * For example, flts32_En4 would have been sfix32_En4 if Data Type Override was
 * off.  This case has power of two scaling, so the fractional slope is the
 * trivial case 1.   For fltu16_S3, the total slope is 3 which is decomposed
 * into Fixed Exponent +1 and Fractional Slope 1.5
 *     When the data type has trivial scaling, including floating point
 * double and single, the total slope is the trivial value 1.
 *   This function will error out if ssGetDataTypeIsFxpFltApiCompat
 * returns false.
 */
FIXPOINT_EXPORT_EXTERN_C double ssGetDataTypeFracSlope(
    SimStruct *S,
    DTypeId dataTypeId
    );

/* Function: ssGetDataTypeFixedExponent ===============================
 *
 * Giving a registered Data Type Id as input, determine the scalings
 * fixed exponent.
 *    S = F * 2^E
 * where
 *   1. <= F < 2.0
 *   S is the Total Slope
 *   F is the Fractional Slope
 *   E is the Fixed Exponent, E is always an integer
 *
 * When the data type a clean binary point interpretation, the Fixed Exponent is
 * simply the negative of the Fraction Length.
 *     When the data type is ScaledDouble, the fixed exponent is determined by
 * what the original data type would  have used if override had not occurred.
 * For example, flts32_En4 would have been sfix32_En4 if Data Type Override was
 * off.  This case has power of two scaling with fraction length +4 and
 * Fixed Exponent -4.   For fltu16_S3, the total slope is 3 which is decomposed
 * into Fixed Exponent +1 and Fractional Slope 1.5
 *     When the data type has trivial scaling, including floating point
 * double and single, the fixed exponent is the trivial value 0.
 *   This function will error out if ssGetDataTypeIsFxpFltApiCompat
 * returns false.
 */
FIXPOINT_EXPORT_EXTERN_C int ssGetDataTypeFixedExponent(
    SimStruct *S,
    DTypeId dataTypeId
    );

FIXPOINT_EXPORT_EXTERN_C void ssFxpConvert(
    SimStruct *S,

    void       *pVoidDest,
    size_t      sizeofDest,
    DTypeId     dataTypeIdDest,

    const void *pVoidSrc,
    size_t      sizeofSrc,
    DTypeId     dataTypeIdSrc,

    fxpModeRounding roundMode,
    fxpModeOverflow overflowMode,

    fxpOverflowLogs *pFxpOverflowLogs
);

FIXPOINT_EXPORT_EXTERN_C double ssFxpConvertToRealWorldValue(
    SimStruct *S,
    const void *pVoidSrc,
    size_t      sizeofSrc,
    DTypeId     dataTypeIdSrc
);

FIXPOINT_EXPORT_EXTERN_C void ssFxpConvertFromRealWorldValue(
    SimStruct *S,

    void       *pVoidDest,
    size_t      sizeofDest,
    DTypeId     dataTypeIdDest,

    double      dblRealWorldValue,

    fxpModeRounding roundMode,
    fxpModeOverflow overflowMode,

    fxpOverflowLogs *pFxpOverflowLogs
);

/* Function ssGetDataTypeNumberOfChunks
 *
 * Giving a dataTypeId as Input, return the number of chunks the container uses.
 *
 */
FIXPOINT_EXPORT_EXTERN_C int ssGetDataTypeNumberOfChunks (
    SimStruct *S,
    DTypeId dataTypeId
    );

/* Function ssFxpGetU32BitRegion
 *
 * This function accesses a fixed point data and returns the stored integer
 * value for the 32 bit region specified by region index. RegionIndex could
 * be any non-negative values. Emulation bits get padded if the RegionIndex
 * is larger than the data size.
 *
 * The input parameters are
 *       pVoid:   a void point to a memory area.
 *       dataTypeId:  a registered fixed point dataTypeId.
 *       regionIndex: the specified 32 bit region.
 *
 * Caution:
 * This function requires dataTypeId to be a valid fixed point data. Floating
 * point data is not supported.
 */
FIXPOINT_EXPORT_EXTERN_C uint32_T ssFxpGetU32BitRegion(
    SimStruct *S,

    const void       *pVoid,

    DTypeId     dataTypeId,

    unsigned int regionIndex
);

/* Function ssFxpSetU32BitRegion
 *
 * This function directly sets the 32 bit region specified by region index for
 * a fixed point data. RegionIndex could be any non-negative values, but only
 * physical bits get written. It will error out if regionValue violates sign
 * extension of the fixed point data.
 *
 * The input parameters are
 *       pVoid:   a void point to a fixed point data.
 *       dataTypeId:  a valid fixed point data type id.
 *       regionValue: the value to be written to the 32 bit region.
 *       regionIndex: the specified 32 bit region.
 *
 * Caution:
 * This function requires dataTypeId to be a valid fixed point data. Floating
 * point data is not supported.
 */
FIXPOINT_EXPORT_EXTERN_C void ssFxpSetU32BitRegion(
    SimStruct *S,

    void       *pVoid,

    DTypeId     dataTypeId,

    uint32_T    regionValue,

    unsigned int regionIndex
);

/* Function: ssLogFixptInstrumentation =============================
 *    Record information collected during simulation, such as
 *    output maximum, minimum, and counts of any overflows, saturations, or
 *    divisions by zero that occurred.
 */
FIXPOINT_EXPORT_EXTERN_C void ssLogFixptInstrumentation(
    SimStruct *S,
    DTypeId dataTypeId,
    double    minValue,
    double    maxValue,
    int countOverflows,
    int countSaturations,
    int countDivisionsByZero,
    char *pStrName
    );

/* Function ssFxpSetU32BitRegionCompliant
 *
 * In a user defined S-Function, if it contains fixed point data type
 * which is larger than 32 bits, it has to call this function to utilize the
 * new memory footprint.
 *
 * The input parameters are:
 *
 *           S:       A point to SimStruct.
 *           Value:   1 means that this S-Function is compliant with new memory footprint.
 *                    0 means that it is not compliant with new memory footprint.
 */
FIXPOINT_EXPORT_EXTERN_C void ssFxpSetU32BitRegionCompliant(
    SimStruct *S,
    int value
);

/* Function ssFxpGetU32BitRegionCompliant
 *
 * This function checks whether the S-Function sets the FxpU32BitRegionCompliant.
 *
 * The input parameters are:
 *
 *           S:       A point to SimStruct.
 *           result:  is the point to returned value.
 */
FIXPOINT_EXPORT_EXTERN_C void ssFxpGetU32BitRegionCompliant(
    SimStruct *S,
    int *result
);

#endif /* fix_published_sfun_api_h */
/* Copyright 1994-2010 The MathWorks, Inc.
 * $Revision: 1.1.8.1 $
 * $Date: 2010/12/15 17:39:54 $
 */

#ifdef SUPPORTS_PRAGMA_ONCE
#pragma once
#endif

#ifndef fix_published_deprecated_h
#define fix_published_deprecated_h

/* Deprecated items provided only for backwards compatibility */

/* The term Doubles-Override is outdated and misleading.
 * Instead, the terms Data-Type-Override and Scaled-Doubles should be used
 * as appropriate.
 * The follow definition is provided for backwards compatibility
 */
#define FXP_STORAGE_DOUBLESOVERRIDE FXP_STORAGE_SCALEDDOUBLE
#define FXP_DT_FIXPT_DBL_OVER FXP_DT_SCALED_DOUBLE
#define fxpIsDataTypeFixPtDblOver(pFxpDataTypeProp)   fxpIsDataTypeScaledDouble(pFxpDataTypeProp)
#define fxpIsDataTypeFloatOrDblOver(pFxpDataTypeProp) fxpIsDataTypeFloatOrSclDbl(pFxpDataTypeProp)

#endif /* fix_published_deprecated_h */
```

### fixpoint_spec.hpp
```cpp
/* Copyright 2008-2011 The MathWorks, Inc. */
/* Generated by genpubheader from export/include/fixpoint/fixpoint_spec.hpp. */

#ifndef FIXPOINT_SPEC_HPP
#define FIXPOINT_SPEC_HPP

#ifdef SUPPORTS_PRAGMA_ONCE
#pragma once
#endif

#ifdef BUILDING_LIBFIXEDPOINT

# define FIXPOINT_EXPORT_CLASS    DLL_EXPORT_SYM
# define FIXPOINT_EXPORT_FCN      DLL_EXPORT_SYM
# define FIXPOINT_EXPORT          DLL_EXPORT_SYM
# define FIXPOINT_EXPORT_EXTERN_C extern "C" DLL_EXPORT_SYM

#elif defined(DLL_IMPORT_SYM)

# define FIXPOINT_EXPORT_CLASS    DLL_IMPORT_SYM
# define FIXPOINT_EXPORT_FCN      DLL_IMPORT_SYM
# define FIXPOINT_EXPORT          DLL_IMPORT_SYM
#ifdef __cplusplus
# define FIXPOINT_EXPORT_EXTERN_C extern "C" DLL_IMPORT_SYM
#else
# define FIXPOINT_EXPORT_EXTERN_C extern DLL_IMPORT_SYM
#endif

#else

#ifdef __cplusplus
#define FIXPOINT_EXPORT_EXTERN_C extern "C"
#else
#define FIXPOINT_EXPORT_EXTERN_C extern
#endif

# define FIXPOINT_EXPORT_CLASS  extern
# define FIXPOINT_EXPORT_FCN    extern
# define FIXPOINT_EXPORT        extern

#endif

#endif
```

### io64.h
```c
/* Copyright 2002-2006 The MathWorks, Inc. */

/* io64.h
 *
 * Include this header file if you need to perform file I/O
 * on large files greater than 2GB (2^31-1 bytes).
 * The definitions in this header file are designed to facilitate
 * cross-platform 64 bit file I/O.
 *
 * This file must be included before any other include file, at the
 * very top of your source file, even before system include files
 * such as stdio.h, to enable 64 bit file I/O for mex files.
 *
 * After including this file (io64.h), you should use the following
 * functions, structs and types for file I/O to enable file I/O beyond
 * the 2GB (2^31-1 byte) limit:
 *
 * fopen()        - 64 bit capable after including this file, use as always
 *                  with no changes
 *
 * getFilePos()   - use this function instead of ftell(), as ftell() is
 *                  not supported for 64 bit file I/O on most platforms.
 *                  getFilePos() is an alias for the POSIX fgetpos()
 *
 * setFilePos()   - use this function instead of fseek(), as fseek() is
 *                  not supported for 64 bit file I/O on most platforms.
 *                  setFilePos() is an alias for the POSIX fsetpos()
 *
 * fpos_T         - the offset argument for getFilePos() and setFilePos()
 *                  is really a pointer to a signed 64 bit integer,
 *                  int64_T, but it must be cast to (fpos_T*)
 *
 * getFileStat()  - use this function instead of stat() to get the size
 *                  in bytes of a file on disk specified by name
 *
 * getFileFstat() - use this function instead of fstat() to get the size
 *                  in bytes of an opened file specified by a FILE* pointer
 *
 * structStat     - use a pointer to a structStat instead of a pointer to
 *                  struct stat as argument to getFileStat() and
 *                  getFileFstat()
 *
 * No changes are required for the following functions:
 *
 * fprintf(), fscanf(), fread(), fwrite(), fclose().
 */

#ifndef __tmw__io64__h__
#define __tmw__io64__h__

#define TMW_ENABLE_INT64 (-1)

/* linux, hpux - must be defined before any other include file */
#if defined(__linux__)
#	undef  _LARGEFILE64_SOURCE
#	define _LARGEFILE64_SOURCE
#endif

#include <stdio.h>
#include <sys/stat.h>

#if defined(_WIN32) /* windows */
#	define getFilePos   fgetpos
#	define setFilePos   fsetpos
#	define structStat   struct _stati64
#	define getFileStat  _stati64
#	define getFileFstat _fstati64
#	define fileno       _fileno
#	define fpos_T       fpos_t
#elif defined(__APPLE__) /* mac */
#	define getFilePos   fgetpos
#	define setFilePos   fsetpos
#	define structStat   struct stat
#	define getFileStat  stat
#	define getFileFstat fstat
#	define fpos_T       fpos_t
#elif defined(__linux__) || defined(__sun)
#	if defined(__GNUC__) && (__GNUC__ >= 3)
		/* fopen works for large files as-is */
#	else
#		define fopen fopen64
#	endif
#	define getFilePos   fgetpos64
#	define setFilePos   fsetpos64
#	define structStat   struct stat64
#	define getFileStat  stat64
#	define getFileFstat fstat64
#	define fpos_T       fpos64_t
#endif

#endif /* __tmw__io64__h__ */
```
